(* PLC project cb_ctud, Dassault Systèmes ControlBuild 2024x *)
(* stored: creationDateTime 2023-10-03T11:12:45-01:00 *)

(* This is a IEC 1131-3 counter /decounter *)
FUNCTION_BLOCK timers_counters.cb_ctud
  VAR_INPUT
    CU : BOOL := false;
    CD : BOOL := false;
    R : BOOL := false;
    LOAD : BOOL := false;
    PV : INT := 0;
  END_VAR
  VAR_OUTPUT
    QU : BOOL := false;
    QD : BOOL := false;
    CV : INT := 0;
  END_VAR


ACTION C_source_code:
/* -----------------------------------------------------------------	*/
/* Type : BFU									*/
/* Copyright : Geensoft							*/
/* Version : 1.1 23/03/2010							*/
/* -----------------------------------------------------------------	*/
/* This is a Up-counter / down-counter	(CTUD)				*/
/* -------------------------------------------------------------	*/
if(R) { CV = 0; }
else {
	if (LOAD) {CV = PV;}
	else {
		if (! (CU && CD)) {
			if(CU && (CV < 32767)) {CV = CV + 1;}
			else {
				if(CD && (CV > -32768)) {CV = CV - 1;}
			}
		}
	}
}
QU = (CV >= PV);
QD = (CV <= 0);
END_ACTION
END_FUNCTION_BLOCK
